// TIA Portal V17 export
// export: Created 2022-06-27T13:56:30.1952817Z, ExportSetting WithDefaults, DisplayName Totally Integrated Automation Portal, DisplayVersion V17 Update 3, DisplayName TIA Portal Openness, DisplayVersion V17 Update 3, DisplayName TIA Portal Version Control Interface, DisplayVersion V17, DisplayName SINAMICS Startdrive Advanced, DisplayVersion V17 Update1, DisplayName SINAMICS Startdrive G110M, G120, G120C, G120D, G120P, G115D, DisplayVersion V17 Update1, DisplayName SINAMICS Startdrive G130, G150, S120, S150, SINAMICS MV, S210, DisplayVersion V17 Update1, DisplayName STEP 7 Professional, DisplayVersion V17 Update 3, DisplayName STEP 7 Safety, DisplayVersion V17, DisplayName WinCC UA Professional, DisplayVersion V17 Update 3
FUNCTION_BLOCK "S0211_CONTROL"   // FB211, LAD
{ S7_Optimized_Access := 'TRUE' }
VERSION : 0.1
// stored: AutoNumber false, IsIECCheckEnabled false, IsRetainMemResEnabled false, MemoryReserve 100, SetENOAutomatically false, UDAEnableTagReadback false
   VAR
      Command : Struct
         ls_bStartproduction : Bool;
         ls_bEnableRoasting : Bool;
         ls_EnableGreenCoffee : Bool;
      END_STRUCT;
      Status : Struct
         ls_bAuto : Bool;
         ls_bStart : Bool;
         ls_bStarting : Bool;
         ls_bRunning : Bool;
         ls_bStopping : Bool;
         ls_bStopped : Bool;
         ls_bHeating : Bool;
         ls_bC1Producing : Bool;
         ls_bC2Producing : Bool;
         ls_iStatusRoaster : Int;
      END_STRUCT;
      HmiData { S7_SetPoint := 'True'} : "pdt_Cmd_Area";
   END_VAR
BEGIN
END_FUNCTION_BLOCK
